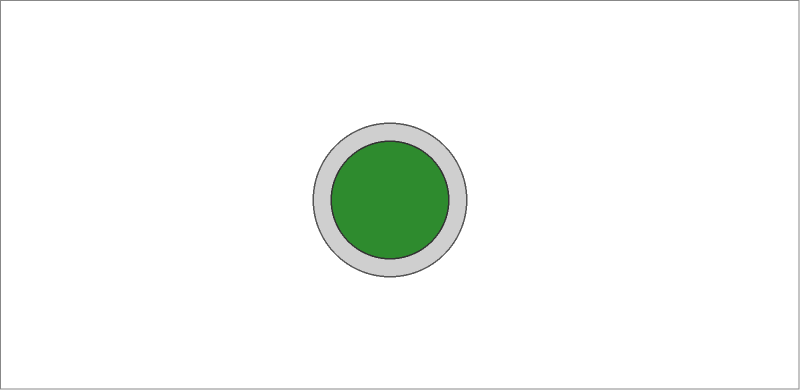
VISUALIZATION VisuDigitalInputControl  // 800x390
VAR_IN_OUT
	fbManualControler	: FB_ManualController ;
END_VAR
    Lamp1 (300,110 180x180), variable: fbManualControler.pDevDigitalInput^.bFcoInputActive, style: Lamp-Lamp1-Green
END_VISUALIZATION

(* stored: Version 1.1.0.1, ProductVersion 3.1.4024.11
   Visu VisuDigitalInputControl: Id {dd63a196-f2d0-0168-23ad-bae36944a229} *)
